{attribute 'qualified_only'}
VAR_GLOBAL
END_VAR

(* stored: Version 1.1.0.1, ProductVersion 3.1.4024.12
   GVL GVL_MotionControl: Id {660c2383-29e1-4473-b80e-34cd4960c117} *)
